// Mitsubishi GX Developer project: パレット取り外し   PLC: Q02

PROGRAM T-PANEL
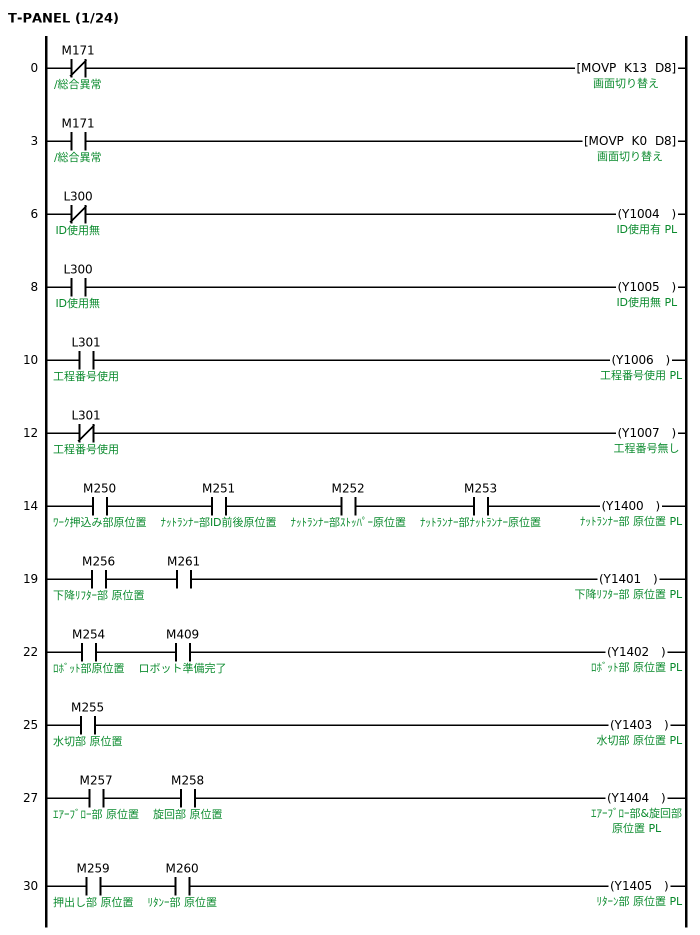
0     LDI     M171  ; /総合異常
      MOVP    K13 D8  ; 画面切り替え
3     LD      M171  ; /総合異常
      MOVP    K0 D8
6     LDI     L300  ; ID使用無
      OUT     Y1004  ; ID使用有 PL
8     LD      L300  ; ID使用無
      OUT     Y1005  ; ID使用無 PL
10    LD      L301  ; 工程番号使用
      OUT     Y1006  ; 工程番号使用 PL
12    LDI     L301  ; 工程番号使用
      OUT     Y1007  ; 工程番号無し
14    LD      M250  ; ﾜｰｸ押込み部原位置
      AND     M251  ; ﾅｯﾄﾗﾝﾅｰ部ID前後原位置
      AND     M252  ; ﾅｯﾄﾗﾝﾅｰ部ｽﾄｯﾊﾟｰ原位置
      AND     M253  ; ﾅｯﾄﾗﾝﾅｰ部ﾅｯﾄﾗﾝﾅｰ原位置
      OUT     Y1400  ; ﾅｯﾄﾗﾝﾅｰ部 原位置 PL
19    LD      M256  ; 下降ﾘﾌﾀｰ部 原位置
      AND     M261
      OUT     Y1401  ; 下降ﾘﾌﾀｰ部 原位置 PL
22    LD      M254  ; ﾛﾎﾞｯﾄ部原位置
      AND     M409  ; ロボット準備完了
      OUT     Y1402  ; ﾛﾎﾞｯﾄ部 原位置 PL
25    LD      M255  ; 水切部 原位置
      OUT     Y1403  ; 水切部 原位置 PL
27    LD      M257  ; ｴｱｰﾌﾞﾛｰ部 原位置
      AND     M258  ; 旋回部 原位置
      OUT     Y1404  ; ｴｱｰﾌﾞﾛｰ部&旋回部 原位置 PL
30    LD      M259  ; 押出し部 原位置
      AND     M260  ; ﾘﾀﾝｰ部 原位置
      OUT     Y1405  ; ﾘﾀｰﾝ部 原位置 PL
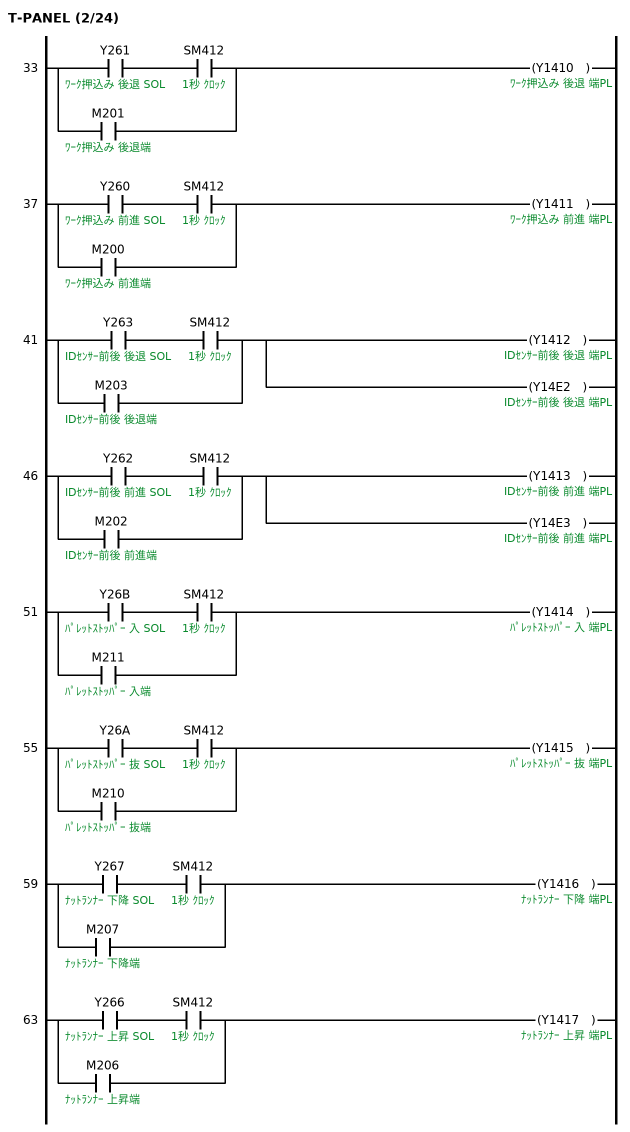
33    LD      Y261  ; ﾜｰｸ押込み 後退 SOL
      AND     SM412  ; 1秒 ｸﾛｯｸ
      OR      M201  ; ﾜｰｸ押込み 後退端
      OUT     Y1410  ; ﾜｰｸ押込み 後退 端PL
37    LD      Y260  ; ﾜｰｸ押込み 前進 SOL
      AND     SM412  ; 1秒 ｸﾛｯｸ
      OR      M200  ; ﾜｰｸ押込み 前進端
      OUT     Y1411  ; ﾜｰｸ押込み 前進 端PL
41    LD      Y263  ; IDｾﾝｻｰ前後 後退 SOL
      AND     SM412  ; 1秒 ｸﾛｯｸ
      OR      M203  ; IDｾﾝｻｰ前後 後退端
      OUT     Y1412  ; IDｾﾝｻｰ前後 後退 端PL
      OUT     Y14E2  ; IDｾﾝｻｰ前後 後退 端PL
46    LD      Y262  ; IDｾﾝｻｰ前後 前進 SOL
      AND     SM412  ; 1秒 ｸﾛｯｸ
      OR      M202  ; IDｾﾝｻｰ前後 前進端
      OUT     Y1413  ; IDｾﾝｻｰ前後 前進 端PL
      OUT     Y14E3  ; IDｾﾝｻｰ前後 前進 端PL
51    LD      Y26B  ; ﾊﾟﾚｯﾄｽﾄｯﾊﾟｰ 入 SOL
      AND     SM412  ; 1秒 ｸﾛｯｸ
      OR      M211  ; ﾊﾟﾚｯﾄｽﾄｯﾊﾟｰ 入端
      OUT     Y1414  ; ﾊﾟﾚｯﾄｽﾄｯﾊﾟｰ 入 端PL
55    LD      Y26A  ; ﾊﾟﾚｯﾄｽﾄｯﾊﾟｰ 抜 SOL
      AND     SM412  ; 1秒 ｸﾛｯｸ
      OR      M210  ; ﾊﾟﾚｯﾄｽﾄｯﾊﾟｰ 抜端
      OUT     Y1415  ; ﾊﾟﾚｯﾄｽﾄｯﾊﾟｰ 抜 端PL
59    LD      Y267  ; ﾅｯﾄﾗﾝﾅｰ 下降 SOL
      AND     SM412  ; 1秒 ｸﾛｯｸ
      OR      M207  ; ﾅｯﾄﾗﾝﾅｰ 下降端
      OUT     Y1416  ; ﾅｯﾄﾗﾝﾅｰ 下降 端PL
63    LD      Y266  ; ﾅｯﾄﾗﾝﾅｰ 上昇 SOL
      AND     SM412  ; 1秒 ｸﾛｯｸ
      OR      M206  ; ﾅｯﾄﾗﾝﾅｰ 上昇端
      OUT     Y1417  ; ﾅｯﾄﾗﾝﾅｰ 上昇 端PL
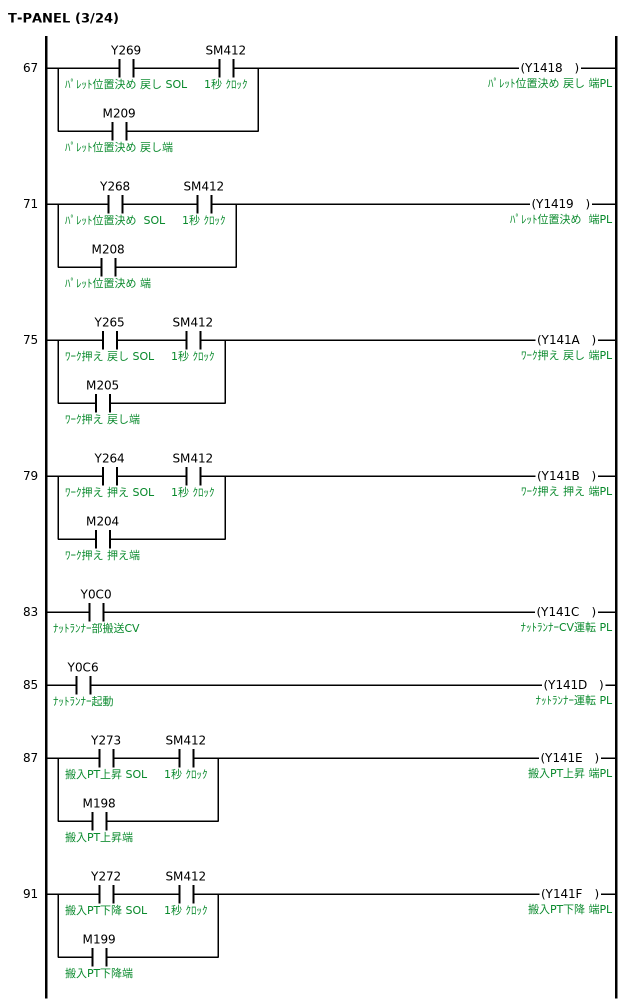
67    LD      Y269  ; ﾊﾟﾚｯﾄ位置決め 戻し SOL
      AND     SM412  ; 1秒 ｸﾛｯｸ
      OR      M209  ; ﾊﾟﾚｯﾄ位置決め 戻し端
      OUT     Y1418  ; ﾊﾟﾚｯﾄ位置決め 戻し 端PL
71    LD      Y268  ; ﾊﾟﾚｯﾄ位置決め  SOL
      AND     SM412  ; 1秒 ｸﾛｯｸ
      OR      M208  ; ﾊﾟﾚｯﾄ位置決め 端
      OUT     Y1419  ; ﾊﾟﾚｯﾄ位置決め  端PL
75    LD      Y265  ; ﾜｰｸ押え 戻し SOL
      AND     SM412  ; 1秒 ｸﾛｯｸ
      OR      M205  ; ﾜｰｸ押え 戻し端
      OUT     Y141A  ; ﾜｰｸ押え 戻し 端PL
79    LD      Y264  ; ﾜｰｸ押え 押え SOL
      AND     SM412  ; 1秒 ｸﾛｯｸ
      OR      M204  ; ﾜｰｸ押え 押え端
      OUT     Y141B  ; ﾜｰｸ押え 押え 端PL
83    LD      Y0C0  ; ﾅｯﾄﾗﾝﾅｰ部搬送CV
      OUT     Y141C  ; ﾅｯﾄﾗﾝﾅｰCV運転 PL
85    LD      Y0C6  ; ﾅｯﾄﾗﾝﾅｰ起動
      OUT     Y141D  ; ﾅｯﾄﾗﾝﾅｰ運転 PL
87    LD      Y273  ; 搬入PT上昇 SOL
      AND     SM412  ; 1秒 ｸﾛｯｸ
      OR      M198  ; 搬入PT上昇端
      OUT     Y141E  ; 搬入PT上昇 端PL
91    LD      Y272  ; 搬入PT下降 SOL
      AND     SM412  ; 1秒 ｸﾛｯｸ
      OR      M199  ; 搬入PT下降端
      OUT     Y141F  ; 搬入PT下降 端PL
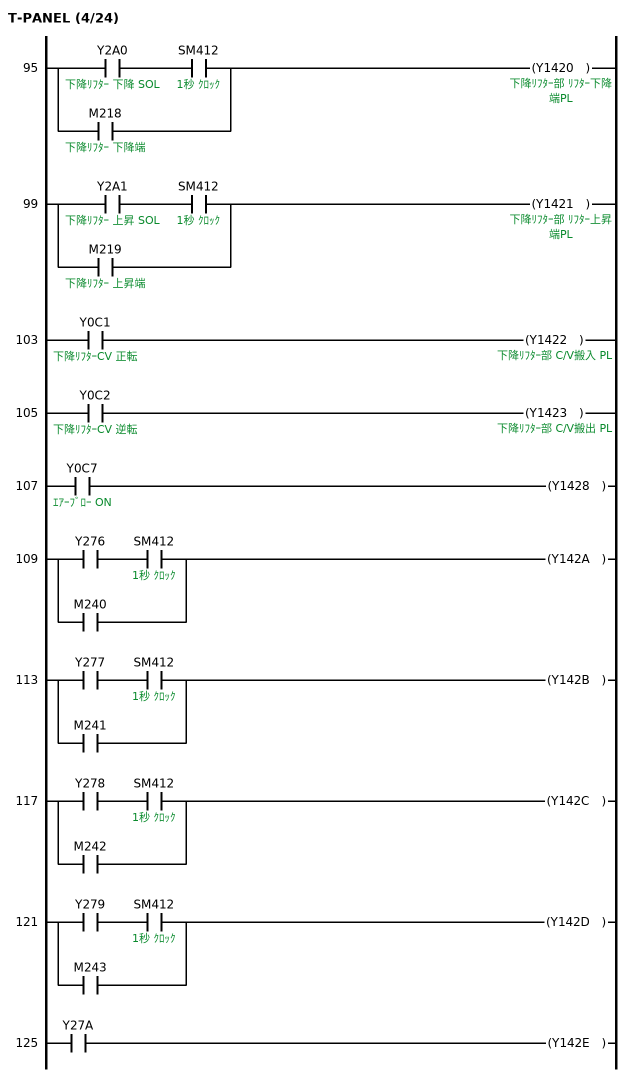
95    LD      Y2A0  ; 下降ﾘﾌﾀｰ 下降 SOL
      AND     SM412  ; 1秒 ｸﾛｯｸ
      OR      M218  ; 下降ﾘﾌﾀｰ 下降端
      OUT     Y1420  ; 下降ﾘﾌﾀｰ部 ﾘﾌﾀｰ下降 端PL
99    LD      Y2A1  ; 下降ﾘﾌﾀｰ 上昇 SOL
      AND     SM412  ; 1秒 ｸﾛｯｸ
      OR      M219  ; 下降ﾘﾌﾀｰ 上昇端
      OUT     Y1421  ; 下降ﾘﾌﾀｰ部 ﾘﾌﾀｰ上昇 端PL
103   LD      Y0C1  ; 下降ﾘﾌﾀｰCV 正転
      OUT     Y1422  ; 下降ﾘﾌﾀｰ部 C/V搬入 PL
105   LD      Y0C2  ; 下降ﾘﾌﾀｰCV 逆転
      OUT     Y1423  ; 下降ﾘﾌﾀｰ部 C/V搬出 PL
107   LD      Y0C7  ; ｴｱｰﾌﾞﾛｰ ON
      OUT     Y1428
109   LD      Y276
      AND     SM412  ; 1秒 ｸﾛｯｸ
      OR      M240
      OUT     Y142A
113   LD      Y277
      AND     SM412  ; 1秒 ｸﾛｯｸ
      OR      M241
      OUT     Y142B
117   LD      Y278
      AND     SM412  ; 1秒 ｸﾛｯｸ
      OR      M242
      OUT     Y142C
121   LD      Y279
      AND     SM412  ; 1秒 ｸﾛｯｸ
      OR      M243
      OUT     Y142D
125   LD      Y27A
      OUT     Y142E
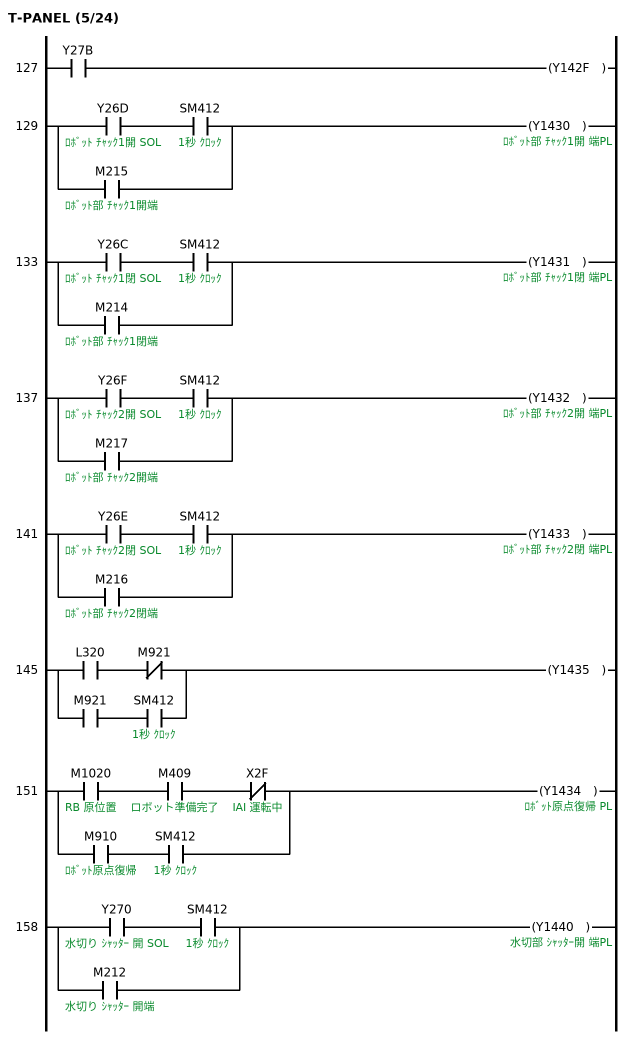
127   LD      Y27B
      OUT     Y142F
129   LD      Y26D  ; ﾛﾎﾞｯﾄ ﾁｬｯｸ1開 SOL
      AND     SM412  ; 1秒 ｸﾛｯｸ
      OR      M215  ; ﾛﾎﾞｯﾄ部 ﾁｬｯｸ1開端
      OUT     Y1430  ; ﾛﾎﾞｯﾄ部 ﾁｬｯｸ1開 端PL
133   LD      Y26C  ; ﾛﾎﾞｯﾄ ﾁｬｯｸ1閉 SOL
      AND     SM412  ; 1秒 ｸﾛｯｸ
      OR      M214  ; ﾛﾎﾞｯﾄ部 ﾁｬｯｸ1閉端
      OUT     Y1431  ; ﾛﾎﾞｯﾄ部 ﾁｬｯｸ1閉 端PL
137   LD      Y26F  ; ﾛﾎﾞｯﾄ ﾁｬｯｸ2開 SOL
      AND     SM412  ; 1秒 ｸﾛｯｸ
      OR      M217  ; ﾛﾎﾞｯﾄ部 ﾁｬｯｸ2開端
      OUT     Y1432  ; ﾛﾎﾞｯﾄ部 ﾁｬｯｸ2開 端PL
141   LD      Y26E  ; ﾛﾎﾞｯﾄ ﾁｬｯｸ2閉 SOL
      AND     SM412  ; 1秒 ｸﾛｯｸ
      OR      M216  ; ﾛﾎﾞｯﾄ部 ﾁｬｯｸ2閉端
      OUT     Y1433  ; ﾛﾎﾞｯﾄ部 ﾁｬｯｸ2閉 端PL
145   LD      L320
      ANI     M921
      LD      M921
      AND     SM412  ; 1秒 ｸﾛｯｸ
      ORB
      OUT     Y1435
151   LD      M1020  ; RB 原位置
      AND     M409  ; ロボット準備完了
      ANI     X2F  ; IAI 運転中
      LD      M910  ; ﾛﾎﾞｯﾄ原点復帰
      AND     SM412  ; 1秒 ｸﾛｯｸ
      ORB
      OUT     Y1434  ; ﾛﾎﾞｯﾄ原点復帰 PL
158   LD      Y270  ; 水切り ｼｬｯﾀｰ 開 SOL
      AND     SM412  ; 1秒 ｸﾛｯｸ
      OR      M212  ; 水切り ｼｬｯﾀｰ 開端
      OUT     Y1440  ; 水切部 ｼｬｯﾀｰ開 端PL
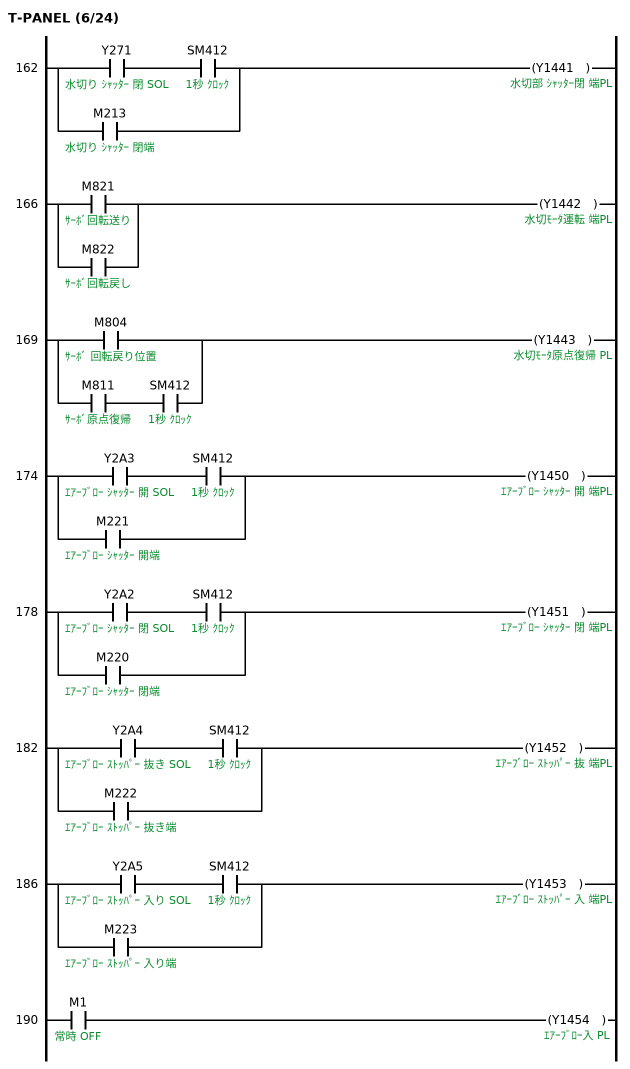
162   LD      Y271  ; 水切り ｼｬｯﾀｰ 閉 SOL
      AND     SM412  ; 1秒 ｸﾛｯｸ
      OR      M213  ; 水切り ｼｬｯﾀｰ 閉端
      OUT     Y1441  ; 水切部 ｼｬｯﾀｰ閉 端PL
166   LD      M821  ; ｻｰﾎﾞ回転送り
      OR      M822  ; ｻｰﾎﾞ回転戻し
      OUT     Y1442  ; 水切ﾓｰﾀ運転 端PL
169   LD      M804  ; ｻｰﾎﾞ 回転戻り位置
      LD      M811  ; ｻｰﾎﾞ原点復帰
      AND     SM412  ; 1秒 ｸﾛｯｸ
      ORB
      OUT     Y1443  ; 水切ﾓｰﾀ原点復帰 PL
174   LD      Y2A3  ; ｴｱｰﾌﾞﾛｰ ｼｬｯﾀｰ 開 SOL
      AND     SM412  ; 1秒 ｸﾛｯｸ
      OR      M221  ; ｴｱｰﾌﾞﾛｰ ｼｬｯﾀｰ 開端
      OUT     Y1450  ; ｴｱｰﾌﾞﾛｰ ｼｬｯﾀｰ 開 端PL
178   LD      Y2A2  ; ｴｱｰﾌﾞﾛｰ ｼｬｯﾀｰ 閉 SOL
      AND     SM412  ; 1秒 ｸﾛｯｸ
      OR      M220  ; ｴｱｰﾌﾞﾛｰ ｼｬｯﾀｰ 閉端
      OUT     Y1451  ; ｴｱｰﾌﾞﾛｰ ｼｬｯﾀｰ 閉 端PL
182   LD      Y2A4  ; ｴｱｰﾌﾞﾛｰ ｽﾄｯﾊﾟｰ 抜き SOL
      AND     SM412  ; 1秒 ｸﾛｯｸ
      OR      M222  ; ｴｱｰﾌﾞﾛｰ ｽﾄｯﾊﾟｰ 抜き端
      OUT     Y1452  ; ｴｱｰﾌﾞﾛｰ ｽﾄｯﾊﾟｰ 抜 端PL
186   LD      Y2A5  ; ｴｱｰﾌﾞﾛｰ ｽﾄｯﾊﾟｰ 入り SOL
      AND     SM412  ; 1秒 ｸﾛｯｸ
      OR      M223  ; ｴｱｰﾌﾞﾛｰ ｽﾄｯﾊﾟｰ 入り端
      OUT     Y1453  ; ｴｱｰﾌﾞﾛｰ ｽﾄｯﾊﾟｰ 入 端PL
190   LD      M1  ; 常時 OFF
      OUT     Y1454  ; ｴｱｰﾌﾞﾛｰ入 PL
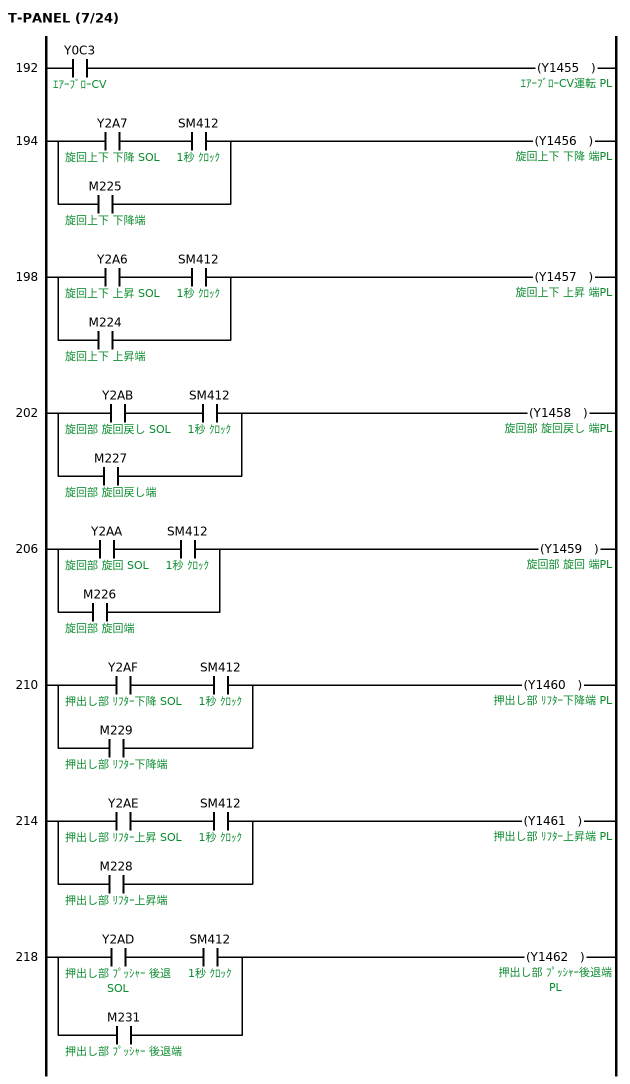
192   LD      Y0C3  ; ｴｱｰﾌﾞﾛｰCV
      OUT     Y1455  ; ｴｱｰﾌﾞﾛｰCV運転 PL
194   LD      Y2A7  ; 旋回上下 下降 SOL
      AND     SM412  ; 1秒 ｸﾛｯｸ
      OR      M225  ; 旋回上下 下降端
      OUT     Y1456  ; 旋回上下 下降 端PL
198   LD      Y2A6  ; 旋回上下 上昇 SOL
      AND     SM412  ; 1秒 ｸﾛｯｸ
      OR      M224  ; 旋回上下 上昇端
      OUT     Y1457  ; 旋回上下 上昇 端PL
202   LD      Y2AB  ; 旋回部 旋回戻し SOL
      AND     SM412  ; 1秒 ｸﾛｯｸ
      OR      M227  ; 旋回部 旋回戻し端
      OUT     Y1458  ; 旋回部 旋回戻し 端PL
206   LD      Y2AA  ; 旋回部 旋回 SOL
      AND     SM412  ; 1秒 ｸﾛｯｸ
      OR      M226  ; 旋回部 旋回端
      OUT     Y1459  ; 旋回部 旋回 端PL
210   LD      Y2AF  ; 押出し部 ﾘﾌﾀｰ下降 SOL
      AND     SM412  ; 1秒 ｸﾛｯｸ
      OR      M229  ; 押出し部 ﾘﾌﾀｰ下降端
      OUT     Y1460  ; 押出し部 ﾘﾌﾀｰ下降端 PL
214   LD      Y2AE  ; 押出し部 ﾘﾌﾀｰ上昇 SOL
      AND     SM412  ; 1秒 ｸﾛｯｸ
      OR      M228  ; 押出し部 ﾘﾌﾀｰ上昇端
      OUT     Y1461  ; 押出し部 ﾘﾌﾀｰ上昇端 PL
218   LD      Y2AD  ; 押出し部 ﾌﾟｯｼｬｰ 後退 SOL
      AND     SM412  ; 1秒 ｸﾛｯｸ
      OR      M231  ; 押出し部 ﾌﾟｯｼｬｰ 後退端
      OUT     Y1462  ; 押出し部 ﾌﾟｯｼｬｰ後退端 PL
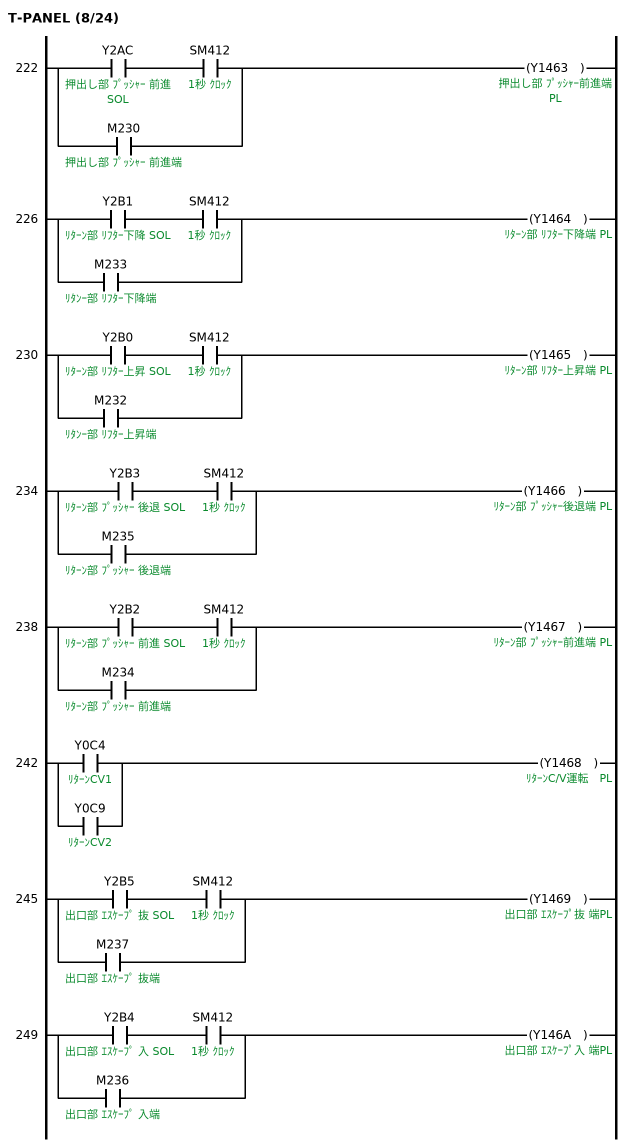
222   LD      Y2AC  ; 押出し部 ﾌﾟｯｼｬｰ 前進 SOL
      AND     SM412  ; 1秒 ｸﾛｯｸ
      OR      M230  ; 押出し部 ﾌﾟｯｼｬｰ 前進端
      OUT     Y1463  ; 押出し部 ﾌﾟｯｼｬｰ前進端 PL
226   LD      Y2B1  ; ﾘﾀｰﾝ部 ﾘﾌﾀｰ下降 SOL
      AND     SM412  ; 1秒 ｸﾛｯｸ
      OR      M233  ; ﾘﾀﾝｰ部 ﾘﾌﾀｰ下降端
      OUT     Y1464  ; ﾘﾀｰﾝ部 ﾘﾌﾀｰ下降端 PL
230   LD      Y2B0  ; ﾘﾀｰﾝ部 ﾘﾌﾀｰ上昇 SOL
      AND     SM412  ; 1秒 ｸﾛｯｸ
      OR      M232  ; ﾘﾀﾝｰ部 ﾘﾌﾀｰ上昇端
      OUT     Y1465  ; ﾘﾀｰﾝ部 ﾘﾌﾀｰ上昇端 PL
234   LD      Y2B3  ; ﾘﾀｰﾝ部 ﾌﾟｯｼｬｰ 後退 SOL
      AND     SM412  ; 1秒 ｸﾛｯｸ
      OR      M235  ; ﾘﾀｰﾝ部 ﾌﾟｯｼｬｰ 後退端
      OUT     Y1466  ; ﾘﾀｰﾝ部 ﾌﾟｯｼｬｰ後退端 PL
238   LD      Y2B2  ; ﾘﾀｰﾝ部 ﾌﾟｯｼｬｰ 前進 SOL
      AND     SM412  ; 1秒 ｸﾛｯｸ
      OR      M234  ; ﾘﾀｰﾝ部 ﾌﾟｯｼｬｰ 前進端
      OUT     Y1467  ; ﾘﾀｰﾝ部 ﾌﾟｯｼｬｰ前進端 PL
242   LD      Y0C4  ; ﾘﾀｰﾝCV1
      OR      Y0C9  ; ﾘﾀｰﾝCV2
      OUT     Y1468  ; ﾘﾀｰﾝC/V運転　PL
245   LD      Y2B5  ; 出口部 ｴｽｹｰﾌﾟ 抜 SOL
      AND     SM412  ; 1秒 ｸﾛｯｸ
      OR      M237  ; 出口部 ｴｽｹｰﾌﾟ 抜端
      OUT     Y1469  ; 出口部 ｴｽｹｰﾌﾟ抜 端PL
249   LD      Y2B4  ; 出口部 ｴｽｹｰﾌﾟ 入 SOL
      AND     SM412  ; 1秒 ｸﾛｯｸ
      OR      M236  ; 出口部 ｴｽｹｰﾌﾟ 入端
      OUT     Y146A  ; 出口部 ｴｽｹｰﾌﾟ入 端PL
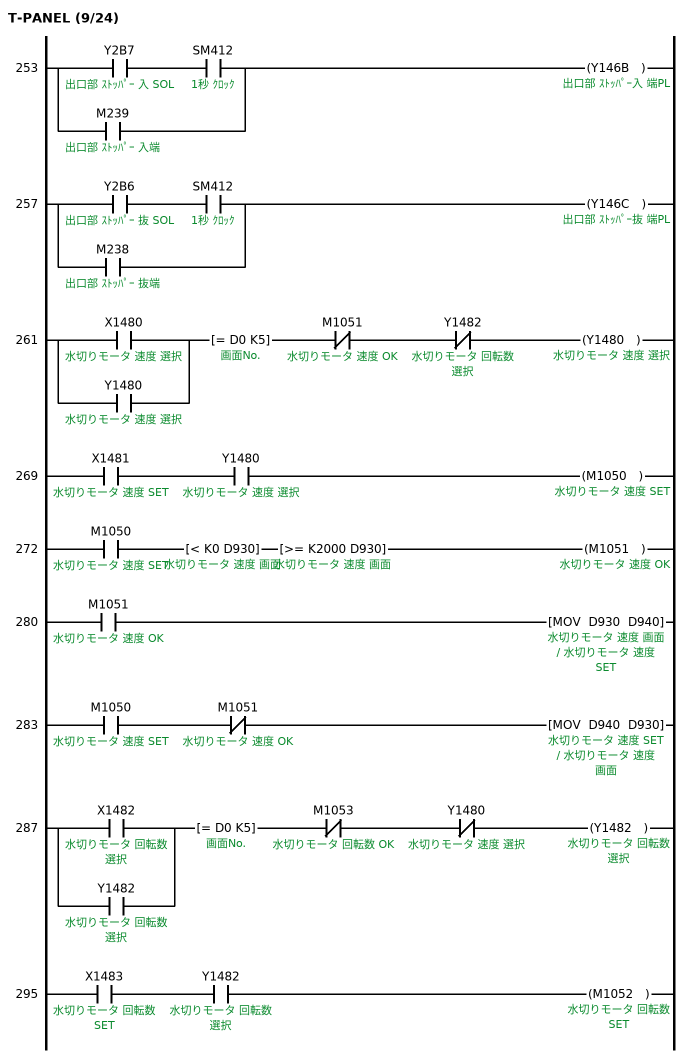
253   LD      Y2B7  ; 出口部 ｽﾄｯﾊﾟｰ 入 SOL
      AND     SM412  ; 1秒 ｸﾛｯｸ
      OR      M239  ; 出口部 ｽﾄｯﾊﾟｰ 入端
      OUT     Y146B  ; 出口部 ｽﾄｯﾊﾟｰ入 端PL
257   LD      Y2B6  ; 出口部 ｽﾄｯﾊﾟｰ 抜 SOL
      AND     SM412  ; 1秒 ｸﾛｯｸ
      OR      M238  ; 出口部 ｽﾄｯﾊﾟｰ 抜端
      OUT     Y146C  ; 出口部 ｽﾄｯﾊﾟｰ抜 端PL
261   LD      X1480  ; 水切りモータ 速度 選択
      OR      Y1480  ; 水切りモータ 速度 選択
      AND=    D0 K5  ; 画面No.
      ANI     M1051  ; 水切りモータ 速度 OK
      ANI     Y1482  ; 水切りモータ 回転数 選択
      OUT     Y1480  ; 水切りモータ 速度 選択
269   LD      X1481  ; 水切りモータ 速度 SET
      AND     Y1480  ; 水切りモータ 速度 選択
      OUT     M1050  ; 水切りモータ 速度 SET
272   LD      M1050  ; 水切りモータ 速度 SET
      AND<    K0 D930  ; 水切りモータ 速度 画面
      AND>=   K2000 D930  ; 水切りモータ 速度 画面
      OUT     M1051  ; 水切りモータ 速度 OK
280   LD      M1051  ; 水切りモータ 速度 OK
      MOV     D930 D940  ; 水切りモータ 速度 SET
283   LD      M1050  ; 水切りモータ 速度 SET
      ANI     M1051  ; 水切りモータ 速度 OK
      MOV     D940 D930
287   LD      X1482  ; 水切りモータ 回転数 選択
      OR      Y1482  ; 水切りモータ 回転数 選択
      AND=    D0 K5  ; 画面No.
      ANI     M1053  ; 水切りモータ 回転数 OK
      ANI     Y1480  ; 水切りモータ 速度 選択
      OUT     Y1482  ; 水切りモータ 回転数 選択
295   LD      X1483  ; 水切りモータ 回転数 SET
      AND     Y1482  ; 水切りモータ 回転数 選択
      OUT     M1052  ; 水切りモータ 回転数 SET
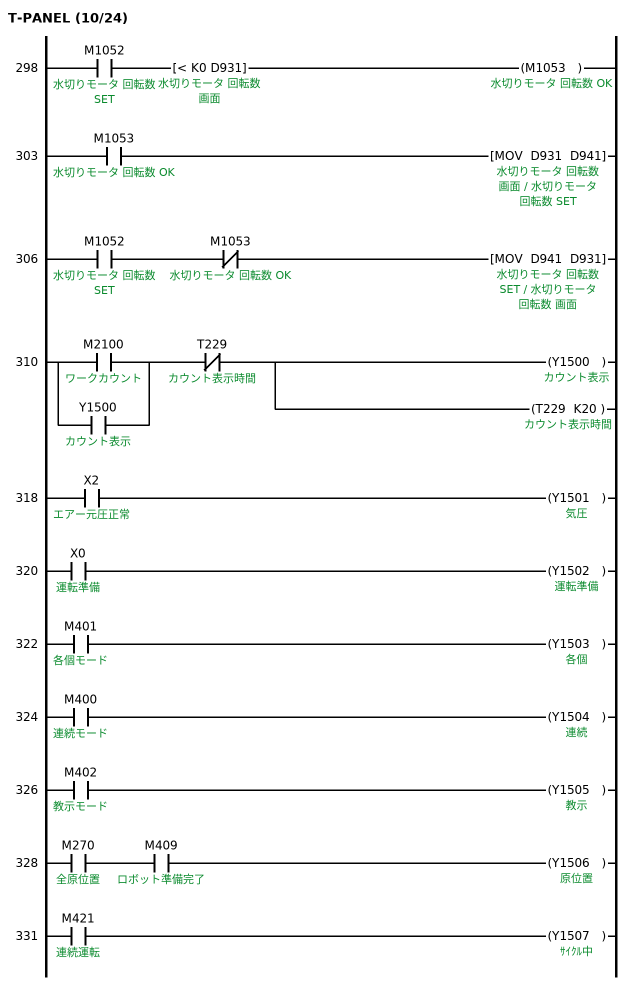
298   LD      M1052  ; 水切りモータ 回転数 SET
      AND<    K0 D931  ; 水切りモータ 回転数 画面
      OUT     M1053  ; 水切りモータ 回転数 OK
303   LD      M1053  ; 水切りモータ 回転数 OK
      MOV     D931 D941  ; 水切りモータ 回転数 SET
306   LD      M1052  ; 水切りモータ 回転数 SET
      ANI     M1053  ; 水切りモータ 回転数 OK
      MOV     D941 D931
310   LD      M2100  ; ワークカウント
      OR      Y1500  ; カウント表示
      ANI     T229  ; カウント表示時間
      OUT     Y1500  ; カウント表示
      OUT     T229 K20  ; カウント表示時間
318   LD      X2  ; エアー元圧正常
      OUT     Y1501  ; 気圧
320   LD      X0  ; 運転準備
      OUT     Y1502  ; 運転準備
322   LD      M401  ; 各個モード
      OUT     Y1503  ; 各個
324   LD      M400  ; 連続モード
      OUT     Y1504  ; 連続
326   LD      M402  ; 教示モード
      OUT     Y1505  ; 教示
328   LD      M270  ; 全原位置
      AND     M409  ; ロボット準備完了
      OUT     Y1506  ; 原位置
331   LD      M421  ; 連続運転
      OUT     Y1507  ; ｻｲｸﾙ中
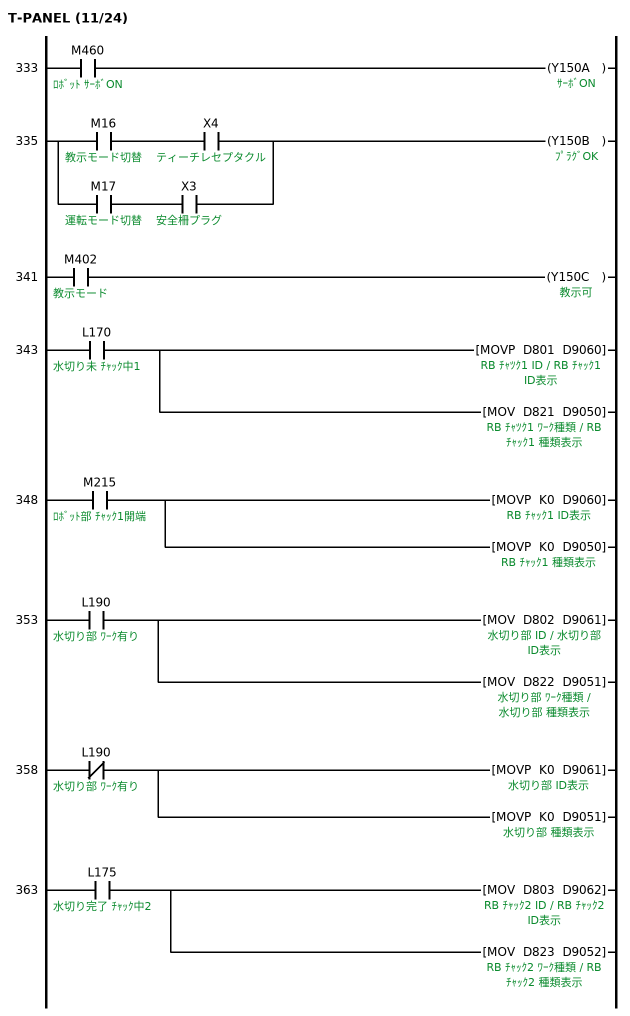
333   LD      M460  ; ﾛﾎﾞｯﾄ ｻｰﾎﾞON
      OUT     Y150A  ; ｻｰﾎﾞON
335   LD      M16  ; 教示モード切替
      AND     X4  ; ティーチレセプタクル
      LD      M17  ; 運転モード切替
      AND     X3  ; 安全柵プラグ
      ORB
      OUT     Y150B  ; ﾌﾟﾗｸﾞOK
341   LD      M402  ; 教示モード
      OUT     Y150C  ; 教示可
343   LD      L170  ; 水切り未 ﾁｬｯｸ中1
      MOVP    D801 D9060  ; RB ﾁｬﾂｸ1 ID / RB ﾁｬｯｸ1 ID表示
      MOV     D821 D9050  ; RB ﾁｬﾂｸ1 ﾜｰｸ種類 / RB ﾁｬｯｸ1 種類表示
348   LD      M215  ; ﾛﾎﾞｯﾄ部 ﾁｬｯｸ1開端
      MOVP    K0 D9060
      MOVP    K0 D9050
353   LD      L190  ; 水切り部 ﾜｰｸ有り
      MOV     D802 D9061  ; 水切り部 ID / 水切り部 ID表示
      MOV     D822 D9051  ; 水切り部 ﾜｰｸ種類 / 水切り部 種類表示
358   LDI     L190  ; 水切り部 ﾜｰｸ有り
      MOVP    K0 D9061
      MOVP    K0 D9051
363   LD      L175  ; 水切り完了 ﾁｬｯｸ中2
      MOV     D803 D9062  ; RB ﾁｬｯｸ2 ID / RB ﾁｬｯｸ2 ID表示
      MOV     D823 D9052  ; RB ﾁｬｯｸ2 ﾜｰｸ種類 / RB ﾁｬｯｸ2 種類表示
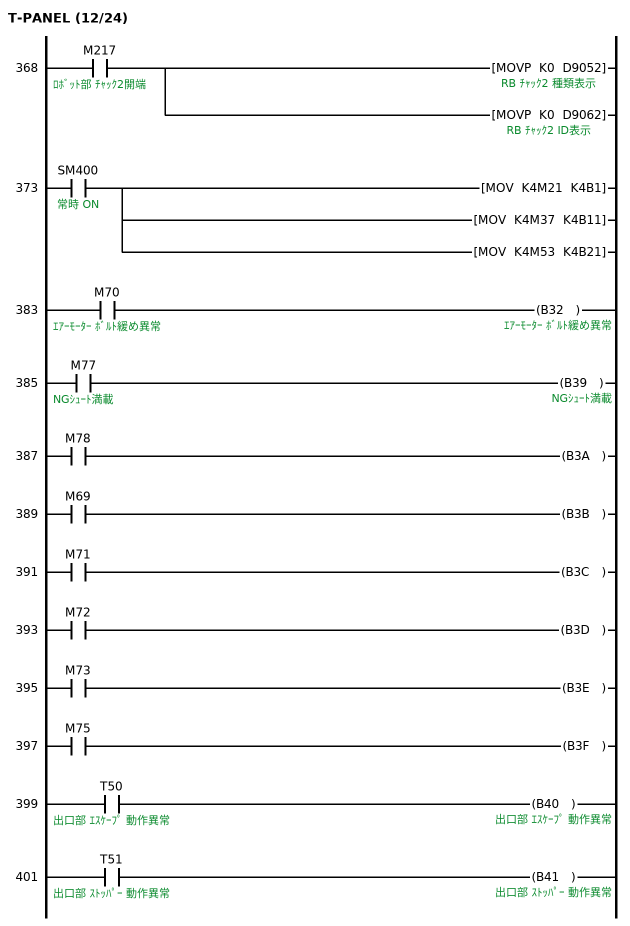
368   LD      M217  ; ﾛﾎﾞｯﾄ部 ﾁｬｯｸ2開端
      MOVP    K0 D9052
      MOVP    K0 D9062
373   LD      SM400  ; 常時 ON
      MOV     K4M21 K4B1  ; PC電池異常 / PC電池異常
      MOV     K4M37 K4B11  ; ﾛﾎﾞｯﾄ部 ﾁｬｯｸ1 LS異常 / ﾛﾎﾞｯﾄ部 ﾁｬｯｸ1 LS異常
      MOV     K4M53 K4B21  ; 下降ﾘﾌﾀｰCV ｻｰﾏﾙﾄﾘｯﾌﾟ / 下降ﾘﾌﾀｰCV ｻｰﾏﾙﾄﾘｯﾌﾟ
383   LD      M70  ; ｴｱｰﾓｰﾀｰ ﾎﾞﾙﾄ緩め異常
      OUT     B32  ; ｴｱｰﾓｰﾀｰ ﾎﾞﾙﾄ緩め異常
385   LD      M77  ; NGｼｭｰﾄ満載
      OUT     B39  ; NGｼｭｰﾄ満載
387   LD      M78
      OUT     B3A
389   LD      M69
      OUT     B3B
391   LD      M71
      OUT     B3C
393   LD      M72
      OUT     B3D
395   LD      M73
      OUT     B3E
397   LD      M75
      OUT     B3F
399   LD      T50  ; 出口部 ｴｽｹｰﾌﾟ 動作異常
      OUT     B40  ; 出口部 ｴｽｹｰﾌﾟ 動作異常
401   LD      T51  ; 出口部 ｽﾄｯﾊﾟｰ 動作異常
      OUT     B41  ; 出口部 ｽﾄｯﾊﾟｰ 動作異常
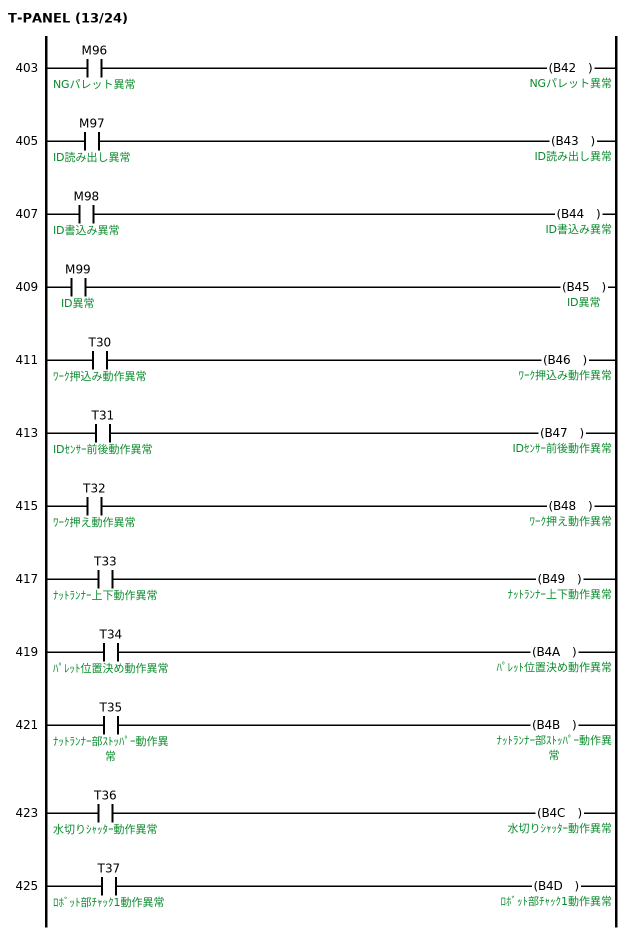
403   LD      M96  ; NGパレット異常
      OUT     B42  ; NGパレット異常
405   LD      M97  ; ID読み出し異常
      OUT     B43  ; ID読み出し異常
407   LD      M98  ; ID書込み異常
      OUT     B44  ; ID書込み異常
409   LD      M99  ; ID異常
      OUT     B45  ; ID異常
411   LD      T30  ; ﾜｰｸ押込み動作異常
      OUT     B46  ; ﾜｰｸ押込み動作異常
413   LD      T31  ; IDｾﾝｻｰ前後動作異常
      OUT     B47  ; IDｾﾝｻｰ前後動作異常
415   LD      T32  ; ﾜｰｸ押え動作異常
      OUT     B48  ; ﾜｰｸ押え動作異常
417   LD      T33  ; ﾅｯﾄﾗﾝﾅｰ上下動作異常
      OUT     B49  ; ﾅｯﾄﾗﾝﾅｰ上下動作異常
419   LD      T34  ; ﾊﾟﾚｯﾄ位置決め動作異常
      OUT     B4A  ; ﾊﾟﾚｯﾄ位置決め動作異常
421   LD      T35  ; ﾅｯﾄﾗﾝﾅｰ部ｽﾄｯﾊﾟｰ動作異常
      OUT     B4B  ; ﾅｯﾄﾗﾝﾅｰ部ｽﾄｯﾊﾟｰ動作異常
423   LD      T36  ; 水切りｼｬｯﾀｰ動作異常
      OUT     B4C  ; 水切りｼｬｯﾀｰ動作異常
425   LD      T37  ; ﾛﾎﾞｯﾄ部ﾁｬｯｸ1動作異常
      OUT     B4D  ; ﾛﾎﾞｯﾄ部ﾁｬｯｸ1動作異常
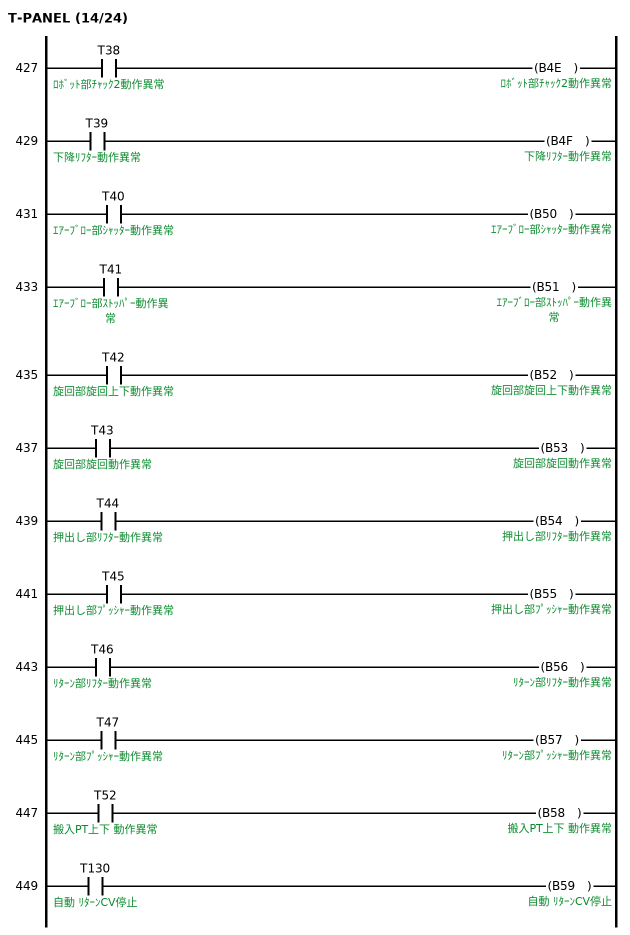
427   LD      T38  ; ﾛﾎﾞｯﾄ部ﾁｬｯｸ2動作異常
      OUT     B4E  ; ﾛﾎﾞｯﾄ部ﾁｬｯｸ2動作異常
429   LD      T39  ; 下降ﾘﾌﾀｰ動作異常
      OUT     B4F  ; 下降ﾘﾌﾀｰ動作異常
431   LD      T40  ; ｴｱｰﾌﾞﾛｰ部ｼｬｯﾀｰ動作異常
      OUT     B50  ; ｴｱｰﾌﾞﾛｰ部ｼｬｯﾀｰ動作異常
433   LD      T41  ; ｴｱｰﾌﾞﾛｰ部ｽﾄｯﾊﾟｰ動作異常
      OUT     B51  ; ｴｱｰﾌﾞﾛｰ部ｽﾄｯﾊﾟｰ動作異常
435   LD      T42  ; 旋回部旋回上下動作異常
      OUT     B52  ; 旋回部旋回上下動作異常
437   LD      T43  ; 旋回部旋回動作異常
      OUT     B53  ; 旋回部旋回動作異常
439   LD      T44  ; 押出し部ﾘﾌﾀｰ動作異常
      OUT     B54  ; 押出し部ﾘﾌﾀｰ動作異常
441   LD      T45  ; 押出し部ﾌﾟｯｼｬｰ動作異常
      OUT     B55  ; 押出し部ﾌﾟｯｼｬｰ動作異常
443   LD      T46  ; ﾘﾀｰﾝ部ﾘﾌﾀｰ動作異常
      OUT     B56  ; ﾘﾀｰﾝ部ﾘﾌﾀｰ動作異常
445   LD      T47  ; ﾘﾀｰﾝ部ﾌﾟｯｼｬｰ動作異常
      OUT     B57  ; ﾘﾀｰﾝ部ﾌﾟｯｼｬｰ動作異常
447   LD      T52  ; 搬入PT上下 動作異常
      OUT     B58  ; 搬入PT上下 動作異常
449   LD      T130  ; 自動 ﾘﾀｰﾝCV停止
      OUT     B59  ; 自動 ﾘﾀｰﾝCV停止
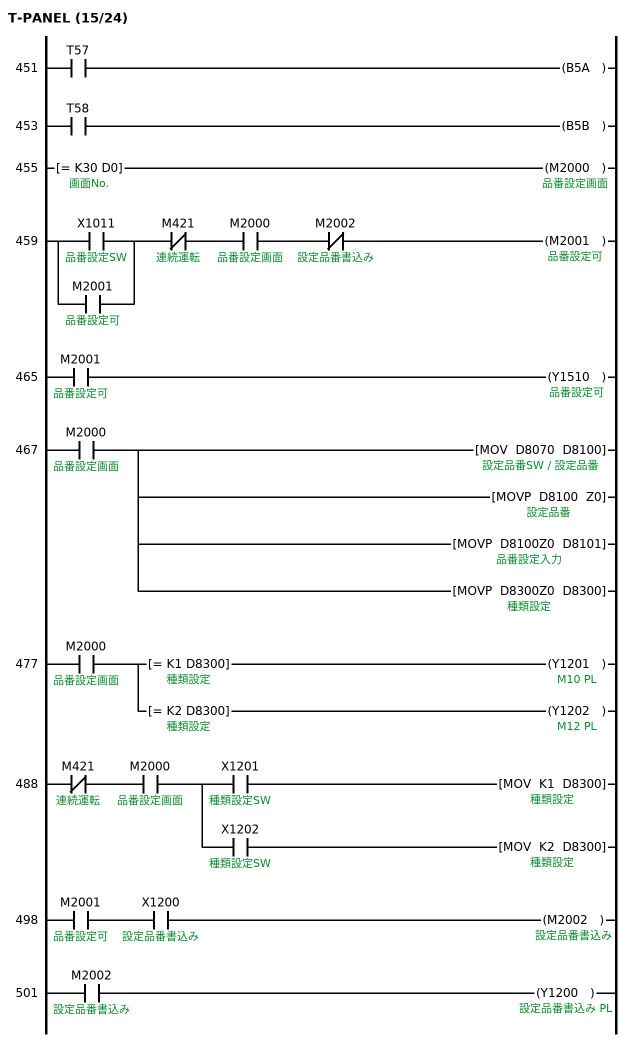
451   LD      T57
      OUT     B5A
453   LD      T58
      OUT     B5B
455   LD=     K30 D0  ; 画面No.
      OUT     M2000  ; 品番設定画面
459   LD      X1011  ; 品番設定SW
      OR      M2001  ; 品番設定可
      ANI     M421  ; 連続運転
      AND     M2000  ; 品番設定画面
      ANI     M2002  ; 設定品番書込み
      OUT     M2001  ; 品番設定可
465   LD      M2001  ; 品番設定可
      OUT     Y1510  ; 品番設定可
467   LD      M2000  ; 品番設定画面
      MOV     D8070 D8100  ; 設定品番SW / 設定品番
      MOVP    D8100 Z0
      MOVP    D8100Z0 D8101  ; 品番設定入力
      MOVP    D8300Z0 D8300  ; 種類設定
477   LD      M2000  ; 品番設定画面
      MPS
      AND=    K1 D8300  ; 種類設定
      OUT     Y1201  ; M10 PL
      MPP
      AND=    K2 D8300  ; 種類設定
      OUT     Y1202  ; M12 PL
488   LDI     M421  ; 連続運転
      AND     M2000  ; 品番設定画面
      MPS
      AND     X1201  ; 種類設定SW
      MOV     K1 D8300
      MPP
      AND     X1202  ; 種類設定SW
      MOV     K2 D8300
498   LD      M2001  ; 品番設定可
      AND     X1200  ; 設定品番書込み
      OUT     M2002  ; 設定品番書込み
501   LD      M2002  ; 設定品番書込み
      OUT     Y1200  ; 設定品番書込み PL
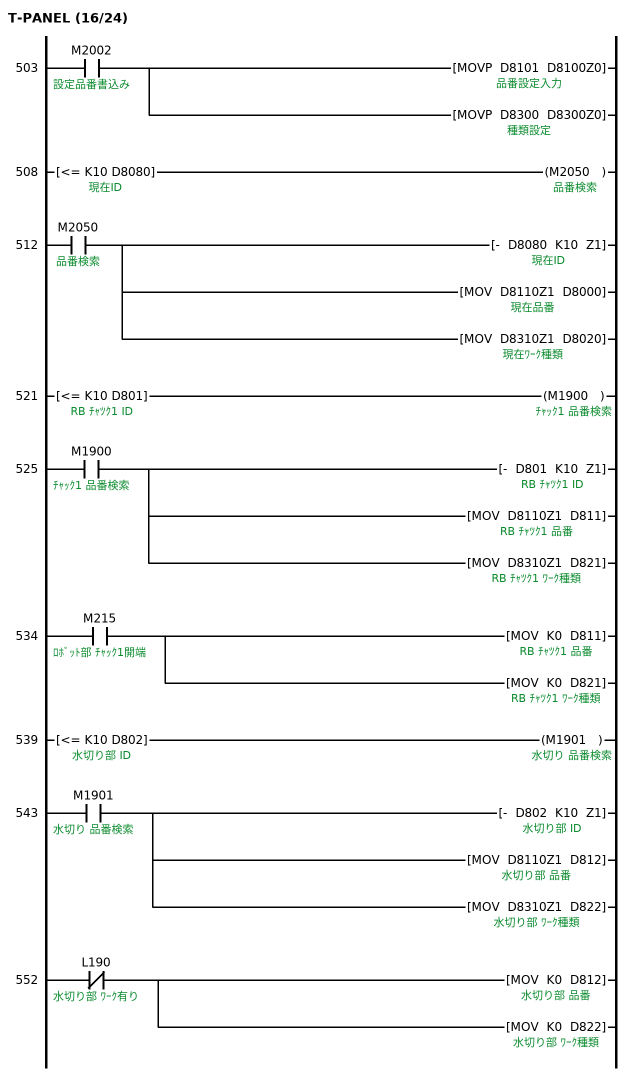
503   LD      M2002  ; 設定品番書込み
      MOVP    D8101 D8100Z0
      MOVP    D8300 D8300Z0
508   LD<=    K10 D8080  ; 現在ID
      OUT     M2050  ; 品番検索
512   LD      M2050  ; 品番検索
      -       D8080 K10 Z1
      MOV     D8110Z1 D8000  ; 現在品番
      MOV     D8310Z1 D8020  ; 現在ﾜｰｸ種類
521   LD<=    K10 D801  ; RB ﾁｬﾂｸ1 ID
      OUT     M1900  ; ﾁｬｯｸ1 品番検索
525   LD      M1900  ; ﾁｬｯｸ1 品番検索
      -       D801 K10 Z1
      MOV     D8110Z1 D811  ; RB ﾁｬﾂｸ1 品番
      MOV     D8310Z1 D821
534   LD      M215  ; ﾛﾎﾞｯﾄ部 ﾁｬｯｸ1開端
      MOV     K0 D811
      MOV     K0 D821
539   LD<=    K10 D802  ; 水切り部 ID
      OUT     M1901  ; 水切り 品番検索
543   LD      M1901  ; 水切り 品番検索
      -       D802 K10 Z1
      MOV     D8110Z1 D812  ; 水切り部 品番
      MOV     D8310Z1 D822
552   LDI     L190  ; 水切り部 ﾜｰｸ有り
      MOV     K0 D812
      MOV     K0 D822
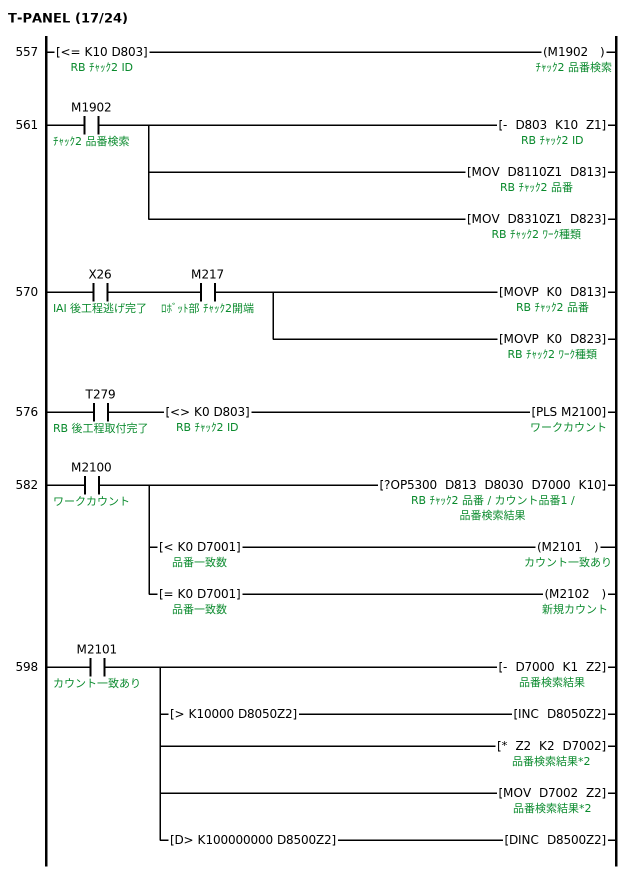
557   LD<=    K10 D803  ; RB ﾁｬｯｸ2 ID
      OUT     M1902  ; ﾁｬｯｸ2 品番検索
561   LD      M1902  ; ﾁｬｯｸ2 品番検索
      -       D803 K10 Z1
      MOV     D8110Z1 D813  ; RB ﾁｬｯｸ2 品番
      MOV     D8310Z1 D823
570   LD      X26  ; IAI 後工程逃げ完了
      AND     M217  ; ﾛﾎﾞｯﾄ部 ﾁｬｯｸ2開端
      MOVP    K0 D813
      MOVP    K0 D823
576   LD      T279  ; RB 後工程取付完了
      AND<>   K0 D803  ; RB ﾁｬｯｸ2 ID
      PLS     M2100  ; ワークカウント
582   LD      M2100  ; ワークカウント
      ?OP5300 D813 D8030 D7000 K10  ; カウント品番1 / 品番検索結果
      MPS
      AND<    K0 D7001  ; 品番一致数
      OUT     M2101  ; カウント一致あり
      MPP
      AND=    K0 D7001  ; 品番一致数
      OUT     M2102  ; 新規カウント
598   LD      M2101  ; カウント一致あり
      -       D7000 K1 Z2
      MPS
      AND>    K10000 D8050Z2
      INC     D8050Z2
      MPP
      *       Z2 K2 D7002  ; 品番検索結果*2
      MOV     D7002 Z2
      ANDD>   K100000000 D8500Z2
      DINC    D8500Z2
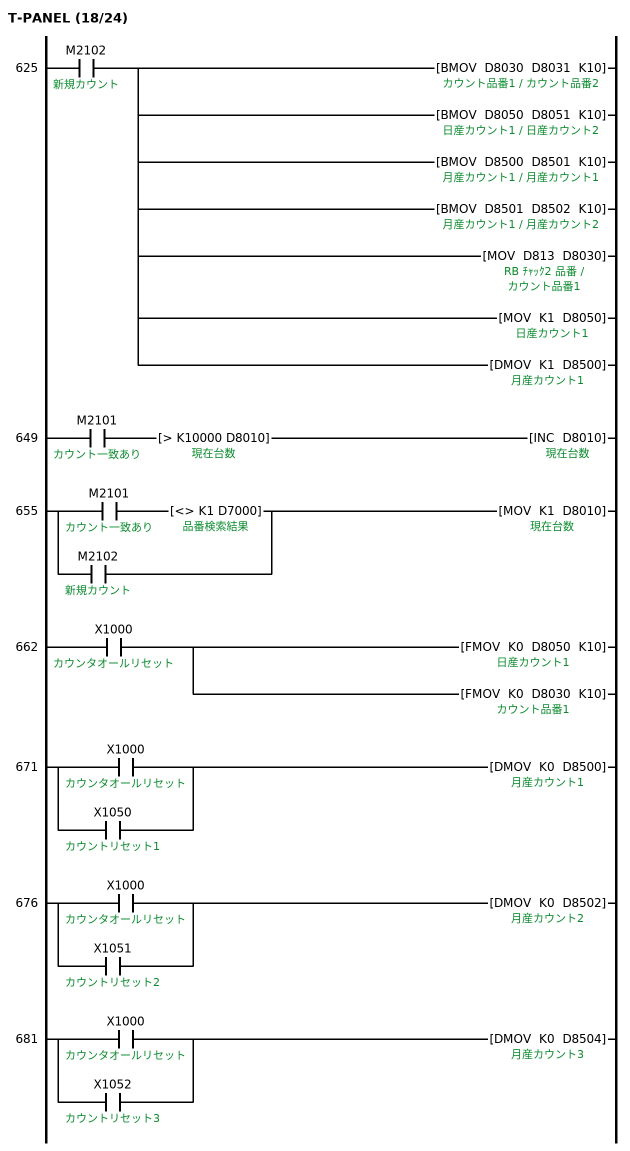
625   LD      M2102  ; 新規カウント
      BMOV    D8030 D8031 K10  ; カウント品番2
      BMOV    D8050 D8051 K10  ; 日産カウント1 / 日産カウント2
      BMOV    D8500 D8501 K10  ; 月産カウント1 / 月産カウント1
      BMOV    D8501 D8502 K10  ; 月産カウント2
      MOV     D813 D8030
      MOV     K1 D8050
      DMOV    K1 D8500
649   LD      M2101  ; カウント一致あり
      AND>    K10000 D8010  ; 現在台数
      INC     D8010
655   LD      M2101  ; カウント一致あり
      AND<>   K1 D7000  ; 品番検索結果
      OR      M2102  ; 新規カウント
      MOV     K1 D8010
662   LD      X1000  ; カウンタオールリセット
      FMOV    K0 D8050 K10
      FMOV    K0 D8030 K10
671   LD      X1000  ; カウンタオールリセット
      OR      X1050  ; カウントリセット1
      DMOV    K0 D8500
676   LD      X1000  ; カウンタオールリセット
      OR      X1051  ; カウントリセット2
      DMOV    K0 D8502
681   LD      X1000  ; カウンタオールリセット
      OR      X1052  ; カウントリセット3
      DMOV    K0 D8504  ; 月産カウント3
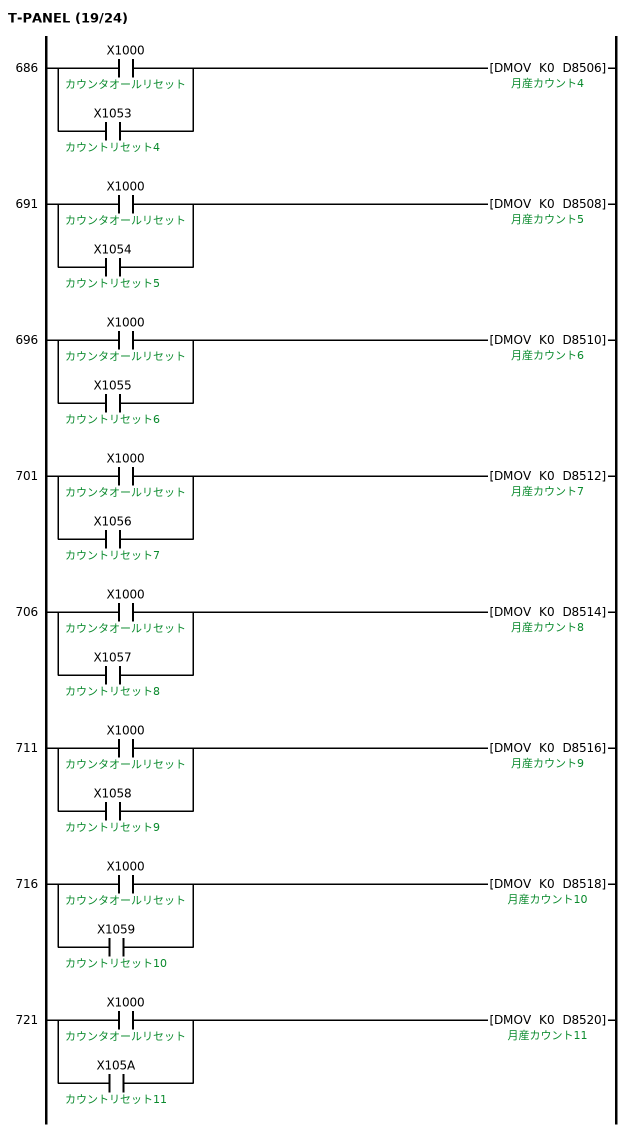
686   LD      X1000  ; カウンタオールリセット
      OR      X1053  ; カウントリセット4
      DMOV    K0 D8506  ; 月産カウント4
691   LD      X1000  ; カウンタオールリセット
      OR      X1054  ; カウントリセット5
      DMOV    K0 D8508  ; 月産カウント5
696   LD      X1000  ; カウンタオールリセット
      OR      X1055  ; カウントリセット6
      DMOV    K0 D8510  ; 月産カウント6
701   LD      X1000  ; カウンタオールリセット
      OR      X1056  ; カウントリセット7
      DMOV    K0 D8512  ; 月産カウント7
706   LD      X1000  ; カウンタオールリセット
      OR      X1057  ; カウントリセット8
      DMOV    K0 D8514  ; 月産カウント8
711   LD      X1000  ; カウンタオールリセット
      OR      X1058  ; カウントリセット9
      DMOV    K0 D8516  ; 月産カウント9
716   LD      X1000  ; カウンタオールリセット
      OR      X1059  ; カウントリセット10
      DMOV    K0 D8518  ; 月産カウント10
721   LD      X1000  ; カウンタオールリセット
      OR      X105A  ; カウントリセット11
      DMOV    K0 D8520  ; 月産カウント11
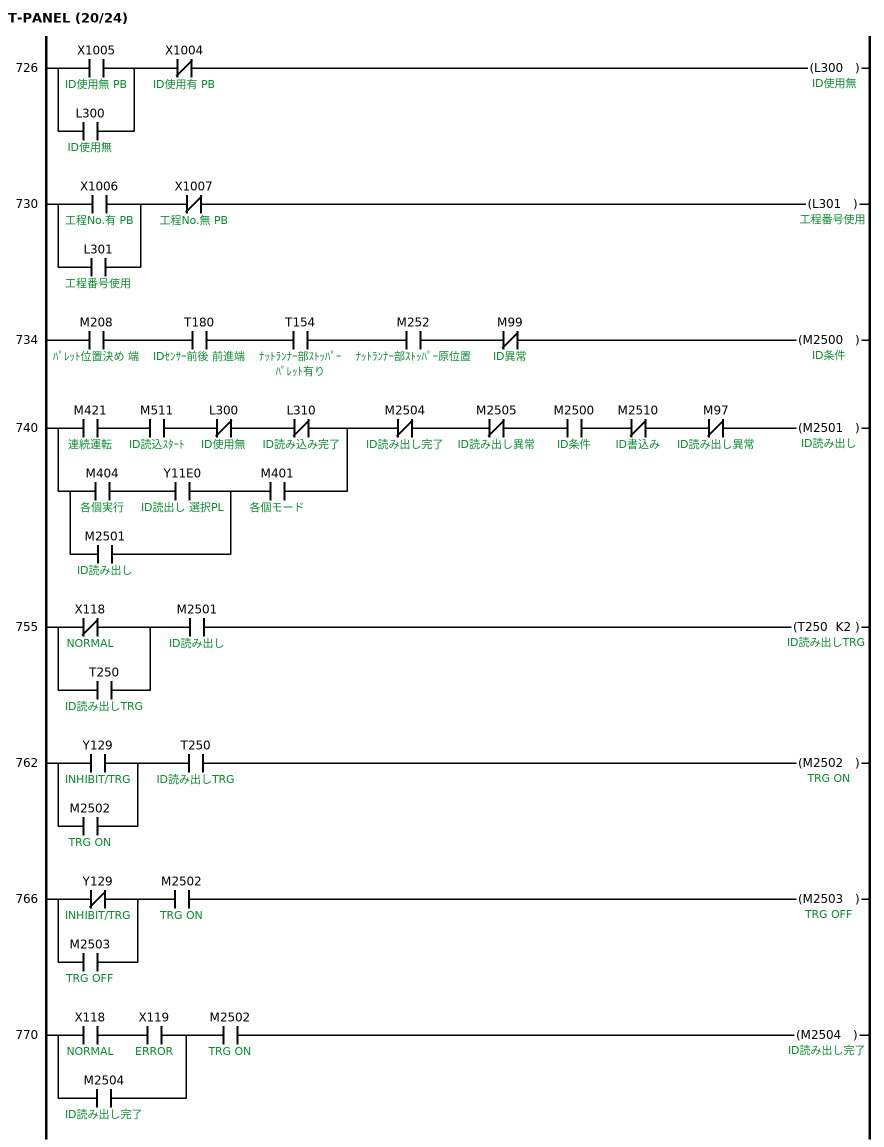
726   LD      X1005  ; ID使用無 PB
      OR      L300  ; ID使用無
      ANI     X1004  ; ID使用有 PB
      OUT     L300  ; ID使用無
730   LD      X1006  ; 工程No.有 PB
      OR      L301  ; 工程番号使用
      ANI     X1007  ; 工程No.無 PB
      OUT     L301  ; 工程番号使用
734   LD      M208  ; ﾊﾟﾚｯﾄ位置決め 端
      AND     T180  ; IDｾﾝｻｰ前後 前進端
      AND     T154  ; ﾅｯﾄﾗﾝﾅｰ部ｽﾄｯﾊﾟｰ ﾊﾟﾚｯﾄ有り
      AND     M252  ; ﾅｯﾄﾗﾝﾅｰ部ｽﾄｯﾊﾟｰ原位置
      ANI     M99  ; ID異常
      OUT     M2500  ; ID条件
740   LD      M421  ; 連続運転
      AND     M511  ; ID読込ｽﾀｰﾄ
      ANI     L300  ; ID使用無
      ANI     L310  ; ID読み込み完了
      LD      M404  ; 各個実行
      AND     Y11E0  ; ID読出し 選択PL
      OR      M2501  ; ID読み出し
      AND     M401  ; 各個モード
      ORB
      ANI     M2504  ; ID読み出し完了
      ANI     M2505  ; ID読み出し異常
      AND     M2500  ; ID条件
      ANI     M2510  ; ID書込み
      ANI     M97  ; ID読み出し異常
      OUT     M2501  ; ID読み出し
755   LDI     X118  ; NORMAL
      OR      T250  ; ID読み出しTRG
      AND     M2501  ; ID読み出し
      OUT     T250 K2  ; ID読み出しTRG
762   LD      Y129  ; INHIBIT/TRG
      OR      M2502  ; TRG ON
      AND     T250  ; ID読み出しTRG
      OUT     M2502  ; TRG ON
766   LDI     Y129  ; INHIBIT/TRG
      OR      M2503  ; TRG OFF
      AND     M2502  ; TRG ON
      OUT     M2503  ; TRG OFF
770   LD      X118  ; NORMAL
      AND     X119  ; ERROR
      OR      M2504  ; ID読み出し完了
      AND     M2502  ; TRG ON
      OUT     M2504  ; ID読み出し完了
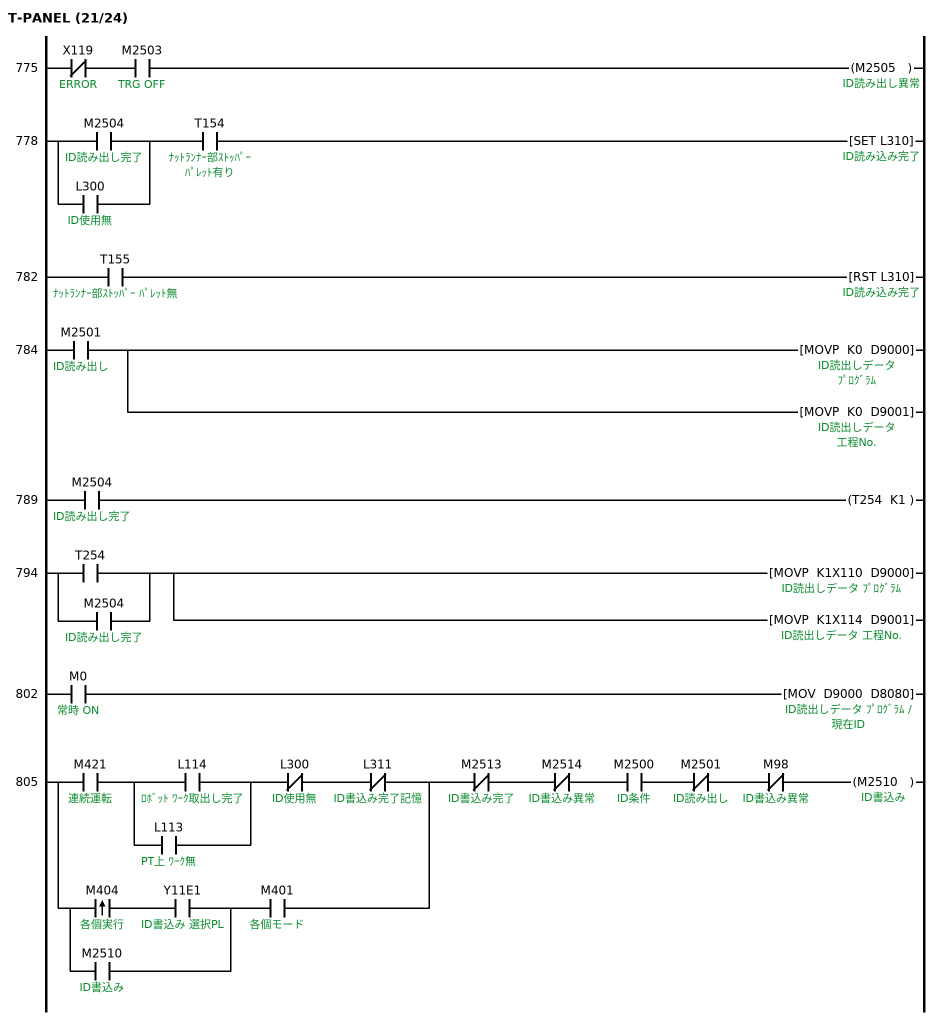
775   LDI     X119  ; ERROR
      AND     M2503  ; TRG OFF
      OUT     M2505  ; ID読み出し異常
778   LD      M2504  ; ID読み出し完了
      OR      L300  ; ID使用無
      AND     T154  ; ﾅｯﾄﾗﾝﾅｰ部ｽﾄｯﾊﾟｰ ﾊﾟﾚｯﾄ有り
      SET     L310  ; ID読み込み完了
782   LD      T155  ; ﾅｯﾄﾗﾝﾅｰ部ｽﾄｯﾊﾟｰ ﾊﾟﾚｯﾄ無
      RST     L310  ; ID読み込み完了
784   LD      M2501  ; ID読み出し
      MOVP    K0 D9000  ; ID読出しデータ ﾌﾟﾛｸﾞﾗﾑ
      MOVP    K0 D9001  ; ID読出しデータ 工程No.
789   LD      M2504  ; ID読み出し完了
      OUT     T254 K1
794   LD      T254
      OR      M2504  ; ID読み出し完了
      MOVP    K1X110 D9000  ; READ DATA 0D0
      MOVP    K1X114 D9001  ; READ DATA 0D4
802   LD      M0  ; 常時 ON
      MOV     D9000 D8080
805   LD      M421  ; 連続運転
      LD      L114  ; ﾛﾎﾞｯﾄ ﾜｰｸ取出し完了
      OR      L113  ; PT上 ﾜｰｸ無
      ANB
      ANI     L300  ; ID使用無
      ANI     L311  ; ID書込み完了記憶
      LDP     M404  ; 各個実行
      AND     Y11E1  ; ID書込み 選択PL
      OR      M2510  ; ID書込み
      AND     M401  ; 各個モード
      ORB
      ANI     M2513  ; ID書込み完了
      ANI     M2514  ; ID書込み異常
      AND     M2500  ; ID条件
      ANI     M2501  ; ID読み出し
      ANI     M98  ; ID書込み異常
      OUT     M2510  ; ID書込み
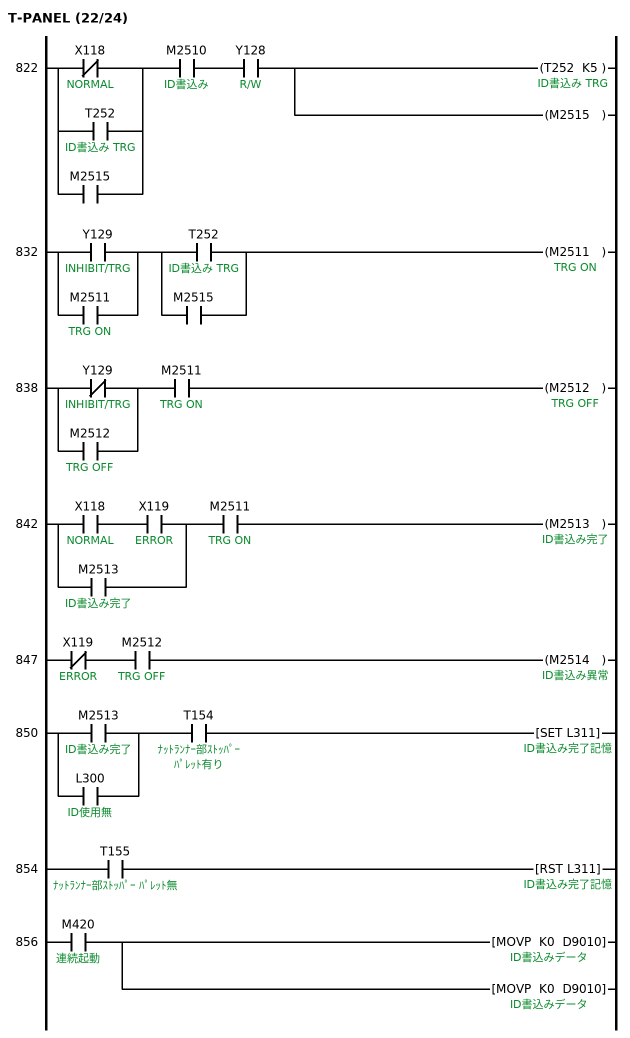
822   LDI     X118  ; NORMAL
      OR      T252  ; ID書込み TRG
      OR      M2515
      AND     M2510  ; ID書込み
      AND     Y128  ; R/W
      OUT     T252 K5  ; ID書込み TRG
      OUT     M2515
832   LD      Y129  ; INHIBIT/TRG
      OR      M2511  ; TRG ON
      LD      T252  ; ID書込み TRG
      OR      M2515
      ANB
      OUT     M2511  ; TRG ON
838   LDI     Y129  ; INHIBIT/TRG
      OR      M2512  ; TRG OFF
      AND     M2511  ; TRG ON
      OUT     M2512  ; TRG OFF
842   LD      X118  ; NORMAL
      AND     X119  ; ERROR
      OR      M2513  ; ID書込み完了
      AND     M2511  ; TRG ON
      OUT     M2513  ; ID書込み完了
847   LDI     X119  ; ERROR
      AND     M2512  ; TRG OFF
      OUT     M2514  ; ID書込み異常
850   LD      M2513  ; ID書込み完了
      OR      L300  ; ID使用無
      AND     T154  ; ﾅｯﾄﾗﾝﾅｰ部ｽﾄｯﾊﾟｰ ﾊﾟﾚｯﾄ有り
      SET     L311  ; ID書込み完了記憶
854   LD      T155  ; ﾅｯﾄﾗﾝﾅｰ部ｽﾄｯﾊﾟｰ ﾊﾟﾚｯﾄ無
      RST     L311  ; ID書込み完了記憶
856   LD      M420  ; 連続起動
      MOVP    K0 D9010  ; ID書込みデータ
      MOVP    K0 D9010
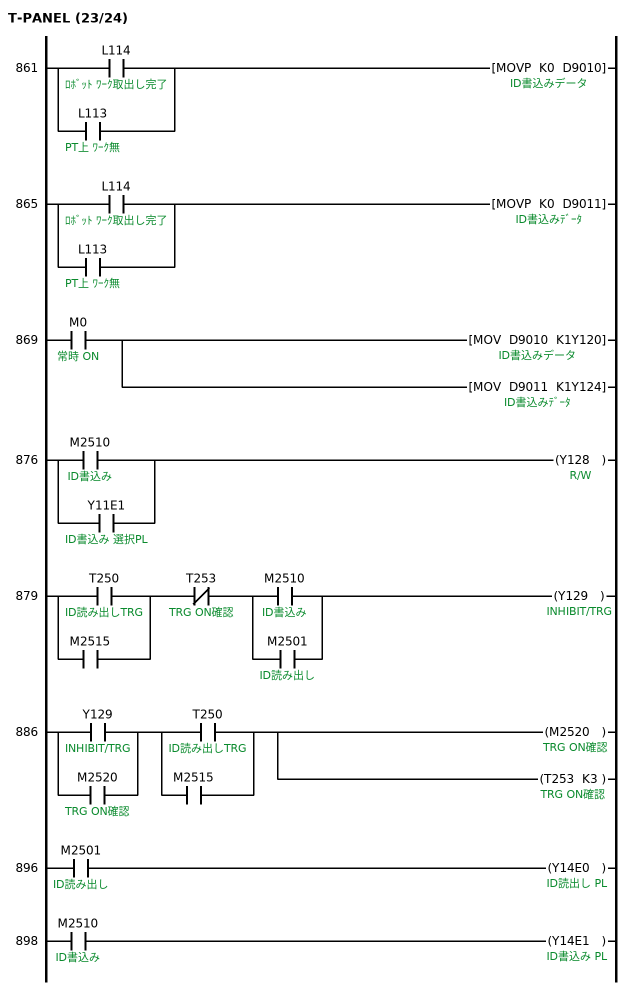
861   LD      L114  ; ﾛﾎﾞｯﾄ ﾜｰｸ取出し完了
      OR      L113  ; PT上 ﾜｰｸ無
      MOVP    K0 D9010
865   LD      L114  ; ﾛﾎﾞｯﾄ ﾜｰｸ取出し完了
      OR      L113  ; PT上 ﾜｰｸ無
      MOVP    K0 D9011  ; ID書込みﾃﾞｰﾀ
869   LD      M0  ; 常時 ON
      MOV     D9010 K1Y120  ; WRITE DATA ID0
      MOV     D9011 K1Y124  ; WRITE DATA ID4
876   LD      M2510  ; ID書込み
      OR      Y11E1  ; ID書込み 選択PL
      OUT     Y128  ; R/W
879   LD      T250  ; ID読み出しTRG
      OR      M2515
      ANI     T253  ; TRG ON確認
      LD      M2510  ; ID書込み
      OR      M2501  ; ID読み出し
      ANB
      OUT     Y129  ; INHIBIT/TRG
886   LD      Y129  ; INHIBIT/TRG
      OR      M2520  ; TRG ON確認
      LD      T250  ; ID読み出しTRG
      OR      M2515
      ANB
      OUT     M2520  ; TRG ON確認
      OUT     T253 K3  ; TRG ON確認
896   LD      M2501  ; ID読み出し
      OUT     Y14E0  ; ID読出し PL
898   LD      M2510  ; ID書込み
      OUT     Y14E1  ; ID書込み PL
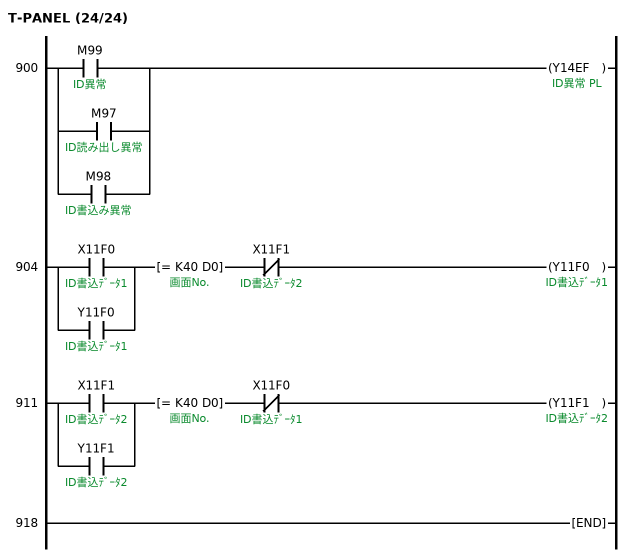
900   LD      M99  ; ID異常
      OR      M97  ; ID読み出し異常
      OR      M98  ; ID書込み異常
      OUT     Y14EF  ; ID異常 PL
904   LD      X11F0  ; ID書込ﾃﾞｰﾀ1
      OR      Y11F0  ; ID書込ﾃﾞｰﾀ1
      AND=    K40 D0  ; 画面No.
      ANI     X11F1  ; ID書込ﾃﾞｰﾀ2
      OUT     Y11F0  ; ID書込ﾃﾞｰﾀ1
911   LD      X11F1  ; ID書込ﾃﾞｰﾀ2
      OR      Y11F1  ; ID書込ﾃﾞｰﾀ2
      AND=    K40 D0  ; 画面No.
      ANI     X11F0  ; ID書込ﾃﾞｰﾀ1
      OUT     Y11F1  ; ID書込ﾃﾞｰﾀ2
918   END
END_PROGRAM
